// TIA Portal V20 export
DATA_BLOCK "MEASLOG_HIST"   // DB44
{ S7_Optimized_Access := 'FALSE' }
VERSION : 0.1
// 표준 접근 : 외부 S7 통신(gr-console) 읽기용. 64 KB 제한으로 MEASLOG 에서 분리
// stored: AutoNumber true, DBAccessibleFromOPCUA true, DBAccessibleFromWebserver true, IsOnlyStoredInLoadMemory false, IsWriteProtectedInAS false
   VAR RETAIN
      LayoutSig : DWord := 16#B320_BA18;   // 레이아웃 서명 (gr-contract gen-sig 가 생성, 수동 수정 금지)
      Entry { S7_SetPoint := 'True'} : Array[0.."MEAS_LOG_LAST"] of "LGR_MeasureLog";   // 측정 이력 (모든 종류, 시간순 링버퍼. 위치는 "MEASLOG".Head/Count/Total)
   END_VAR
BEGIN
   // Entry[0].Data[0] : MeasureItem Status
   // Entry[0].Data[1] : MeasureItem InnerDiameter
   // Entry[0].Data[2] : MeasureItem upperBead Height
   // Entry[0].Data[3] : MeasureItem Item Height
   // Entry[0].Data[4] : MeasureItem
   // Entry[0].Data[5] : MeasureItem
   // Entry[0].Data[6] : MeasureItem
   // Entry[0].Data[7] : MeasureItem Torq InnerDiameter
   // Entry[0].Data[8] : MeasureItem Torq factor
   // Entry[0].Data[9] : MeasureItem
   // Entry[0].Data[10] : MeasureItem Entry InnerDiameter
   // Entry[0].Data[11] : MeasureItem Entry upperBead Height
   // Entry[0].Data[12] : MeasureItem Entry Item Height
   // Entry[0].Data[13] : MeasureItem Entry OffsetX
   // Entry[0].Data[14] : MeasureItem Entry OffsetY
   // Entry[0].Data[15] : MeasureItem Exit InnerDiameter
   // Entry[0].Data[16] : MeasureItem Exit upperBead Height
   // Entry[0].Data[17] : MeasureItem Exit Item Height
   // Entry[0].Data[18] : MeasureItem Exit OffsetX
   // Entry[0].Data[19] : MeasureItem Exit OffsetY
END_DATA_BLOCK
